FUNCTION_BLOCK FB_ResetIntegralController
VAR_INPUT
	stParam 				: ST_Parameters;
	fVelocityReference_ms	: LREAL;
	fPositionError_m		: LREAL;
END_VAR
VAR_OUTPUT
	bReset: BOOL;
END_VAR
VAR
END_VAR

IF ABS(fVelocityReference_ms) > 0.0 THEN 
    bReset := FALSE;
ELSIF ABS(fPositionError_m) > stParam.stClosedLoopControlSettings.fMaxPositionError THEN 
    bReset := FALSE;
ELSE 
    bReset := TRUE;
END_IF;

END_FUNCTION_BLOCK

(* stored: Version 1.1.0.1, ProductVersion 3.1.4024.10
   POU FB_ResetIntegralController: Id {0d649c07-5b1e-4f69-9d0d-d4c49aa2a0af}, SpecialFunc None *)
